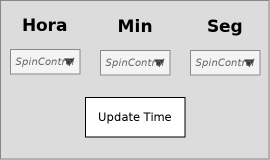
VISUALIZATION Hora  // 270x160
    Rectangle (85,97 100x40), "Update Time"
        tap GVL_TimeSch.bUpdateTime
    SpinControl (10,49 70x25), variable: GVL_TimeSch.timeToInsert.wHour
        OnMouseClick: write the text variable via Default, min 0, max 23
    Label (10,10 70x30), "Hora"
    SpinControl (100,50 70x25), variable: GVL_TimeSch.timeToInsert.wMinute
        OnMouseClick: write the text variable via Default, min 0, max 59
    Label (100,11 70x30), "Min"
    SpinControl (190,50 70x25), variable: GVL_TimeSch.timeToInsert.wSecond
        OnMouseClick: write the text variable via Default, min 0, max 59
    Label (190,11 70x30), "Seg"
END_VISUALIZATION

(* stored: Version 1.1.0.1
   Visu Hora: Id {67d8022f-fc1f-4c71-9cda-2bcdb042b259} *)
